KUKA KRL program: placebox2.src, placebox2.dat

--- placebox2.src ---
&ACCESS RVO1
&COMMENT
&ACCESS RVP
&PARAM EDITMASK = *
&PARAM TEMPLATE = C:\KRC\Roboter\Template\vorgabe
&PARAM DISKPATH = KRC:\R1\Program
DEF placebox2(current_box_layer1:in, current_box_layer_side1:in, X_box:in, Z_box:in, Z_washer:in, Kz_washer1:in, Z_pallet:in)
decl int current_box_layer1, current_box_layer_side1, X_box, Z_box, Z_washer, Kz_washer1, Z_pallet
;current_box_layer1 - number of the current layer of boxes at place 1
;current_box_layer_side1 - number of the side of the placed boxes at place 1. 1 - right side, 2 - left side
;X_box - length of the box, [mm]
del pos XP1m, XP2m, XP3m

; check if there is a requirement to enter the zone from the operator
IF (Entry_Request) THEN
Go_home()
BRAKE
;FOLD WAIT Time= 0.5 sec;%{PE}%R 8.3.22,%MKUKATPBASIS,%CWAIT,%VWAIT,%P 2:0.5
WAIT SEC 0.5
;ENDFOLD
HALT
ENDIF

XP1m = XP1
XP2m = XP2
XP2m.z = XP2.z + Z_pallet*2 ; 200 - height of one pallet
; calculation of Z coordinates of the current layer
XP2m.z = XP2m.z + Z_washer * Kz_washer1 + Z_box * (current_box_layer1 - 1)
XP3m = XP2m
XP3m.z = XP2m.z + 200

; movement to the right or to the left side of the place point
IF (current_box_layer_side1 == 1) THEN
; right side
; calculation of coordinates
XP1m.C = 180
; movement to the point above the place point
;FOLD LIN P1m  Vel=2 m/s CPDAT0 Tool[3]:tool_2_box Base[2]:plpallet1;%{PE}%R 8.3.22,%MKUKATPBASIS,%CMOVE,%VLIN,%P 1:LIN, 2:P1m, 3:, 5:2, 7:CPDAT0
$BWDSTART=FALSE
LDAT_ACT=LCPDAT0
FDAT_ACT=FP1m
BAS(#CP_PARAMS,2)
LIN XP1m
;ENDFOLD
XP2m.C = 180
; movement down to the place point
;FOLD LIN P2m  Vel=2 m/s CPDAT0 Tool[3]:tool_2_box Base[2]:plpallet1;%{PE}%R 8.3.22,%MKUKATPBASIS,%CMOVE,%VLIN,%P 1:LIN, 2:P2m, 3:, 5:2, 7:CPDAT0
$BWDSTART=FALSE
LDAT_ACT=LCPDAT0
FDAT_ACT=FP2m
BAS(#CP_PARAMS,2)
LIN XP2m
;ENDFOLD

; take off the support
;FOLD OUT 2 'support hook right'  State= FALSE;%{PE}%R 8.3.22,%MKUKATPBASIS,%COUT,%VOUTX,%P 2:2, 3:support hook right, 5:FALSE, 6:

$OUT[2]=FALSE
;ENDFOLD
;FOLD OUT 4 'support hook left'  State= FALSE;%{PE}%R 8.3.22,%MKUKATPBASIS,%COUT,%VOUTX,%P 2:4, 3:support hook left, 5:FALSE, 6:

$OUT[4]=FALSE
;ENDFOLD
;FOLD WAIT Time=1 sec;%{PE}%R 8.3.32,%MKUKATPBASIS,%CWAIT,%VWAIT,%P 3:1
WAIT SEC 1
;ENDFOLD

; take off the boxes
;FOLD OUT 1 'finger right'  State= FALSE;%{PE}%R 8.3.22,%MKUKATPBASIS,%COUT,%VOUTX,%P 2:1, 3:finger right, 5:FALSE, 6:

$OUT[1]=FALSE
;ENDFOLD
;FOLD OUT 3 'finger left'  State= FALSE;%{PE}%R 8.3.22,%MKUKATPBASIS,%COUT,%VOUTX,%P 2:3, 3:finger left, 5:FALSE, 6:

$OUT[3]=FALSE
;ENDFOLD
;FOLD WAIT Time= 0.5 sec;%{PE}%R 8.3.22,%MKUKATPBASIS,%CWAIT,%VWAIT,%P 2:0.5
WAIT SEC 0.5
;ENDFOLD

XP3m.C = 180
; movement up
;FOLD LIN P3m  Vel=2 m/s CPDAT0 Tool[2]:tool_empty Base[2]:plpallet1;%{PE}%R 8.3.22,%MKUKATPBASIS,%CMOVE,%VLIN,%P 1:LIN, 2:P3m, 3:, 5:2, 7:CPDAT0
$BWDSTART=FALSE
LDAT_ACT=LCPDAT0
FDAT_ACT=FP3m
BAS(#CP_PARAMS,2)
LIN XP3m
;ENDFOLD

ELSE
IF (current_box_layer_side2 == 2) THEN
; left side
; calculation of coordinates
XP1m.C = -180
XP1m.y = XP1m.y - 200
; movement to the point above the place point
;FOLD LIN P1m  Vel=2 m/s CPDAT0 Tool[3]:tool_2_box Base[2]:plpallet1;%{PE}%R 8.3.22,%MKUKATPBASIS,%CMOVE,%VLIN,%P 1:LIN, 2:P1m, 3:, 5:2, 7:CPDAT0
$BWDSTART=FALSE
LDAT_ACT=LCPDAT0
FDAT_ACT=FP1m
BAS(#CP_PARAMS,2)
LIN XP1m
;ENDFOLD
XP2m.C = -180
XP2m.y = XP2m.y - 200
; movement down to the place point
;FOLD LIN P2m  Vel=2 m/s CPDAT0 Tool[3]:tool_2_box Base[2]:plpallet1;%{PE}%R 8.3.22,%MKUKATPBASIS,%CMOVE,%VLIN,%P 1:LIN, 2:P2m, 3:, 5:2, 7:CPDAT0
$BWDSTART=FALSE
LDAT_ACT=LCPDAT0
FDAT_ACT=FP2m
BAS(#CP_PARAMS,2)
LIN XP2m
;ENDFOLD

; take off the support
;FOLD OUT 2 'support hook right'  State= FALSE;%{PE}%R 8.3.22,%MKUKATPBASIS,%COUT,%VOUTX,%P 2:2, 3:support hook right, 5:FALSE, 6:

$OUT[2]=FALSE
;ENDFOLD
;FOLD OUT 4 'support hook left'  State= FALSE;%{PE}%R 8.3.22,%MKUKATPBASIS,%COUT,%VOUTX,%P 2:4, 3:support hook left, 5:FALSE, 6:

$OUT[4]=FALSE
;ENDFOLD
;FOLD WAIT Time=1 sec;%{PE}%R 8.3.32,%MKUKATPBASIS,%CWAIT,%VWAIT,%P 3:1
WAIT SEC 1
;ENDFOLD

; take off the boxes
;FOLD OUT 1 'finger right'  State= FALSE;%{PE}%R 8.3.22,%MKUKATPBASIS,%COUT,%VOUTX,%P 2:1, 3:finger right, 5:FALSE, 6:

$OUT[1]=FALSE
;ENDFOLD
;FOLD OUT 3 'finger left'  State= FALSE;%{PE}%R 8.3.22,%MKUKATPBASIS,%COUT,%VOUTX,%P 2:3, 3:finger left, 5:FALSE, 6:

$OUT[3]=FALSE
;ENDFOLD
;FOLD WAIT Time= 0.5 sec;%{PE}%R 8.3.22,%MKUKATPBASIS,%CWAIT,%VWAIT,%P 2:0.5
WAIT SEC 0.5
;ENDFOLD

XP3m.C = -180
; movement up
;FOLD LIN P3m  Vel=2 m/s CPDAT0 Tool[2]:tool_empty Base[2]:plpallet1;%{PE}%R 8.3.22,%MKUKATPBASIS,%CMOVE,%VLIN,%P 1:LIN, 2:P3m, 3:, 5:2, 7:CPDAT0
$BWDSTART=FALSE
LDAT_ACT=LCPDAT0
FDAT_ACT=FP3m
BAS(#CP_PARAMS,2)
LIN XP3m
;ENDFOLD

ENDIF
ENDIF

;check for signal from sensors that upper pallet is now not free
IF (L2_Pallet_2_clear == TRUE) THEN
    $MSG_T.TYP = #quit
    $MSG_T.KEY[]="Signal s datchika, chto verkhn'aya palleta na meste 1 svobodna" ;MSG
    $MSG_T.VALID=TRUE ;vivvod MSG
    ; wait for aknowledgement
    WHILE  $MSG_T.VALID == true
    ; WAIT SEC 0.05
    ENDWHILE
ENDIF
;FOLD WAIT FOR ( L2_Pallet_2_clear  );%{PE}%R 8.3.22,%MKUKATPBASIS,%CEXT_WAIT_FOR,%VEXT_WAIT_FOR,%P 2:, 4:, 5:L2_Pallet_2_clear, 6:1, 7:, 9:
WAIT FOR  (  (L2_Pallet_2_clear) )
;ENDFOLD

; movement up with rotation of the gripper
;FOLD LIN P4  Vel=2 m/s CPDAT4 Tool[2]:tool_empty Base[2]:plpallet1;%{PE}%R 8.3.22,%MKUKATPBASIS,%CMOVE,%VLIN,%P 1:LIN, 2:P4, 3:, 5:2, 7:CPDAT4
$BWDSTART=FALSE
LDAT_ACT=LCPDAT4
FDAT_ACT=FP4
BAS(#CP_PARAMS,2)
LIN XP4
;ENDFOLD

;FOLD PTP home  Vel=100 % PDAT5 Tool[2]:tool_empty Base[0];%{PE}%R 8.3.22,%MKUKATPBASIS,%CMOVE,%VPTP,%P 1:PTP, 2:home, 3:, 5:100, 7:PDAT5
$BWDSTART=FALSE
PDAT_ACT=PPDAT5
FDAT_ACT=Fhome
BAS(#PTP_PARAMS,100)
PTP Xhome
;ENDFOLD

END

--- placebox2.dat ---
&ACCESS RVO1
&COMMENT
DEFDAT placebox2 PUBLIC
;FOLD EXTERNAL DECLARATIONS;%{PE}%MKUKATPBASIS,%CEXT,%VCOMMON,%P
;FOLD BASISTECH EXT;%{PE}%MKUKATPBASIS,%CEXT,%VEXT,%P
EXT  BAS (BAS_COMMAND  :IN,REAL  :IN )
DECL INT SUCCESS
;ENDFOLD (BASISTECH EXT)
;FOLD USER EXT;%{E}%MKUKATPUSER,%CEXT,%VEXT,%P
;Make here your modifications

;ENDFOLD (USER EXT)
;ENDFOLD (EXTERNAL DECLERATIONS)
; DECL BASIS_SUGG_T LAST_BASIS={POINT1[] "home                    ",POINT2[] "home                    ",CP_PARAMS[] "CPDAT3                  ",PTP_PARAMS[] "PDAT4                   ",CONT[] "                        ",CP_VEL[] "2                       ",PTP_VEL[] "100                     ",SYNC_PARAMS[] "SYNCDAT                 ",SPL_NAME[] "S0                      ",A_PARAMS[] "ADAT0                   "}
DECL E6POS XP1={X 13.9638586,Y -2.41177225,Z 747.639282,A 1.16506231,B 0.0120191490,C 179.989105,S 2,T 3,E1 0.0,E2 0.0,E3 0.0,E4 0.0,E5 0.0,E6 0.0}
DECL FDAT FP1={TOOL_NO 0,BASE_NO 0,IPO_FRAME #BASE,POINT2[] "P1",TQ_STATE FALSE}
DECL LDAT LCPDAT1={VEL 2,ACC 100,APO_DIST 100,APO_FAC 50,AXIS_VEL 100.0,AXIS_ACC 100.0,ORI_TYP #VAR,CIRC_TYP #BASE,JERK_FAC 50.0,GEAR_JERK 50.0,EXAX_IGN 0}

DECL LDAT LCPDAT0={VEL 2,ACC 100,APO_DIST 100,APO_FAC 50,AXIS_VEL 100.0,AXIS_ACC 100.0,ORI_TYP #VAR,CIRC_TYP #BASE,JERK_FAC 50.0,GEAR_JERK 50.0,EXAX_IGN 0}
DECL E6POS XP1m={X 1463.90698,Y -2335.81665,Z 678.544678,A 1.96151149,B -8.27161622E-14,C -180.000,S 2,T 3,E1 0.0,E2 0.0,E3 0.0,E4 0.0,E5 0.0,E6 0.0}
DECL FDAT FP1m={TOOL_NO 3,BASE_NO 2,IPO_FRAME #BASE,POINT2[] " ",TQ_STATE FALSE}

DECL E6POS XP2={X 14.1800137,Y -2.20657802,Z -6.12030271E-05,A 1.16514552,B 1.28041397E-14,C 180.000,S 2,T 3,E1 0.0,E2 0.0,E3 0.0,E4 0.0,E5 0.0,E6 0.0}
DECL LDAT LCPDAT2={VEL 2.00000,ACC 100.000,APO_DIST 100.000,APO_FAC 50.0000,AXIS_VEL 100.000,AXIS_ACC 100.000,ORI_TYP #VAR,CIRC_TYP #BASE,JERK_FAC 50.0000,GEAR_JERK 50.0000,EXAX_IGN 0}
DECL PDAT PPDAT2={VEL 100.000,ACC 100.000,APO_DIST 100.000,GEAR_JERK 50.0000}

DECL E6POS XP2m={X 1463.90698,Y -2335.81665,Z 678.544678,A 1.96151149,B -8.27161622E-14,C -180.000,S 2,T 3,E1 0.0,E2 0.0,E3 0.0,E4 0.0,E5 0.0,E6 0.0}
DECL FDAT FP2m={TOOL_NO 3,BASE_NO 2,IPO_FRAME #BASE,POINT2[] " ",TQ_STATE FALSE}

DECL E6POS XP3m={X 1463.90698,Y -2335.81665,Z 678.544678,A 1.96151149,B -8.27161622E-14,C -180.000,S 2,T 3,E1 0.0,E2 0.0,E3 0.0,E4 0.0,E5 0.0,E6 0.0}
DECL FDAT FP3m={TOOL_NO 2,BASE_NO 2,IPO_FRAME #BASE,POINT2[] " ",TQ_STATE FALSE}

DECL BASIS_SUGG_T LAST_BASIS={POINT1[] "P4",POINT2[] "P4",CP_PARAMS[] "CPDAT4",PTP_PARAMS[] "PDAT0",CONT[] " ",CP_VEL[] "2",PTP_VEL[] "100",SYNC_PARAMS[] "e ",SPL_NAME[] "Home "}
DECL E6POS XP4={X 14.1800137,Y -2.20657802,Z 389.601654,A 1.16514552,B 7.20532304E-14,C 180.000,S 2,T 3,E1 0.0,E2 0.0,E3 0.0,E4 0.0,E5 0.0,E6 0.0}

DECL FDAT FP4={TOOL_NO 2,BASE_NO 2,IPO_FRAME #BASE,POINT2[] " ",TQ_STATE FALSE}
DECL LDAT LCPDAT4={VEL 2,ACC 100,APO_DIST 100,APO_FAC 50,AXIS_VEL 100.0,AXIS_ACC 100.0,ORI_TYP #VAR,CIRC_TYP #BASE,JERK_FAC 50.0,GEAR_JERK 50.0,EXAX_IGN 0}

ENDDAT
